{attribute 'qualified_only'}
{attribute 'strict'}
TYPE E_ExternalBrake :
(
    eBrakeClosed := 0,
    eDelayBrakeOpening := 1,
    eBrakeOpened := 2,
    eBrakeCloseDelayAmplifier := 3
);
END_TYPE

(* stored: Version 1.1.0.1
   EnumerationTextList E_ExternalBrake: Id {3b0ef411-d8a7-0ec7-258f-652b9a44dc44} *)
